Omron CX-Programmer project NewProject (CX-Programmer 9.73)

# PLC NewPLC1: CP1E N20

## Global symbols (name address type ; comment)
0.01 BOOL  ; pb start
0.02 BOOL  ; pb stop
0.03 BOOL  ; sensor full
100.01 BOOL  ; open gate
100.02 BOOL  ; cylinder 1
100.04 BOOL  ; gate 2
200.00 BOOL  ; relay
T001 BOOL  ; timer
T002 BOOL  ; timer2

## Program NewProgram1 (cyclic task 0)

### Section Section1

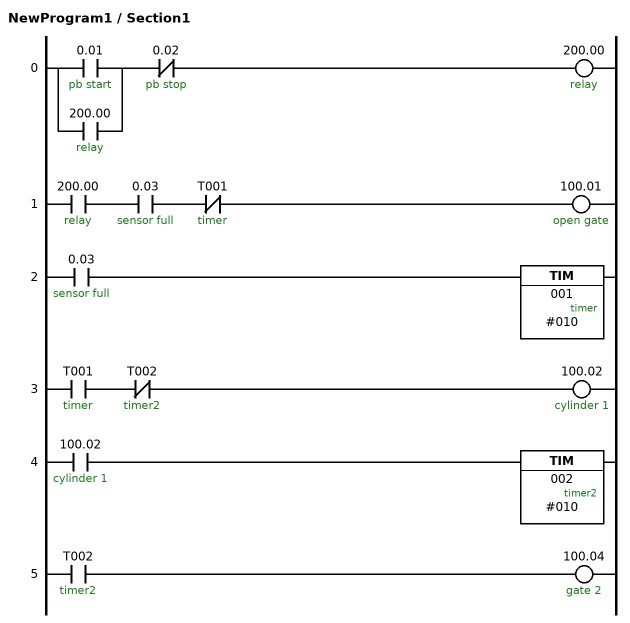
; rung 0
LD 0.01  ; pb start
OR 200.00  ; relay
ANDNOT 0.02  ; pb stop
OUT 200.00  ; relay
; rung 1
LD 200.00  ; relay
AND 0.03  ; sensor full
ANDNOT T001  ; timer
OUT 100.01  ; open gate
; rung 2
LD 0.03  ; sensor full
TIM 001 #010  ; timer
; rung 3
LD T001  ; timer
ANDNOT T002  ; timer2
OUT 100.02  ; cylinder 1
; rung 4
LD 100.02  ; cylinder 1
TIM 002 #010  ; timer2
; rung 5
LD T002  ; timer2
OUT 100.04  ; gate 2

### Section END
; rung 0
END(001)